TYPE Vec4i : ARRAY[1..4] OF INT; END_TYPE

(* stored: Version 1.1.0.1, ProductVersion 3.1.4024.12
   DUT Vec4i: Id {e7b5fa99-7254-46b9-8016-be1d79a9a438} *)
